// TIA Portal V19 export
FUNCTION "A02_HMI_CALL" : Void   // FC228, LAD
// stored: SetENOAutomatically false
BEGIN

REGION Network 1
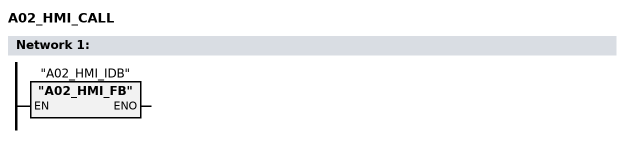
   RUNG wire#powerrail
      "A02_HMI_IDB"()
   END_RUNG
   // the same network as SCL:
   "A02_HMI_IDB"();   // "A02_HMI_FB"
END_REGION
END_FUNCTION
